% RSLogix 500 project Digital Control.RSS, saved by version 8.30.00.16 %
PROJECT "UNTITLED"    % processor: Bul.1763 MicroLogix 1100 Series B %

PROGRAM FILES
  LAD 2   3 rungs
  LAD 3 "IO"  5 rungs
  LAD 4 "CTRL"  11 rungs

DATA FILES
  O0 OUTPUT  4 elements
  I1 INPUT  6 elements
  S2 STATUS  66 elements
  B3 BINARY  1 elements
  T4 TIMER  4 elements
  C5 COUNTER  1 elements
  R6 CONTROL  1 elements
  N7 INTEGER  1 elements
  F8 FLOAT  1 elements

LADDER 2
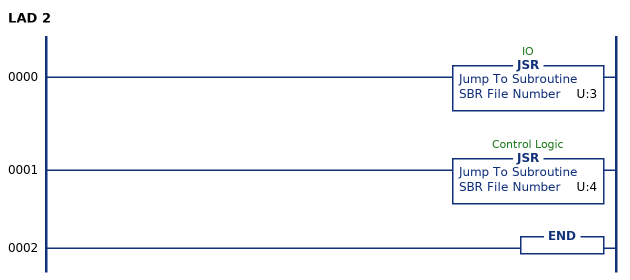
% Rung: 0 %
SOR JSR U:3 EOR
%   U:3  "IO" %
% Rung: 1 %
SOR JSR U:4 EOR
%   U:4  "Control Logic" %
% Rung: 2 %
SOR END EOR

LADDER 3 "IO"
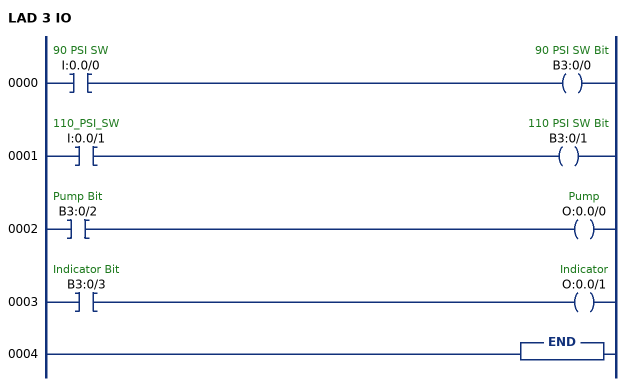
% Rung: 0 %
SOR XIC I:0.0/0 OTE B3:0/0 EOR
%   I:0.0/0  "90 PSI SW" %
%   B3:0/0  "90 PSI SW Bit" %
% Rung: 1 %
SOR XIC I:0.0/1 OTE B3:0/1 EOR
%   I:0.0/1  110_PSI_SW %
%   B3:0/1  "110 PSI SW Bit" %
% Rung: 2 %
SOR XIC B3:0/2 OTE O:0.0/0 EOR
%   B3:0/2  "Pump Bit" %
%   O:0.0/0  "Pump" %
% Rung: 3 %
SOR XIC B3:0/3 OTE O:0.0/1 EOR
%   B3:0/3  "Indicator Bit" %
%   O:0.0/1  "Indicator" %
% Rung: 4 %
SOR END EOR

LADDER 4 "CTRL"
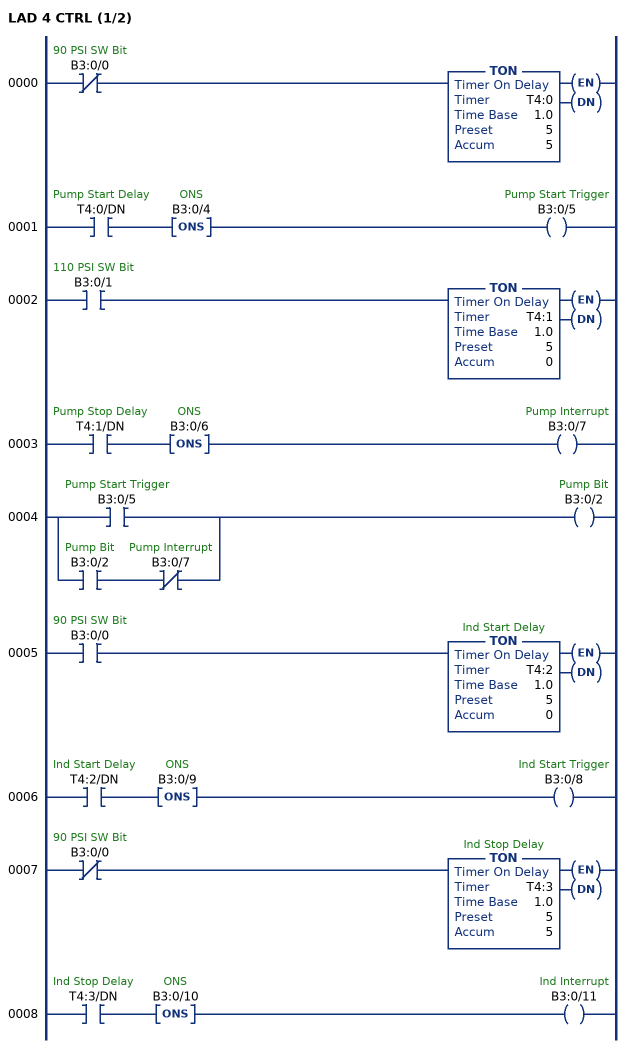
% Rung: 0 %
SOR XIO B3:0/0 TON T4:0 1.0 5 5 EOR
%   B3:0/0  "90 PSI SW Bit" %
% Rung: 1 %
SOR XIC T4:0/DN ONS B3:0/4 OTE B3:0/5 EOR
%   T4:0/DN  "Pump Start Delay" %
%   B3:0/4  "ONS" %
%   B3:0/5  "Pump Start Trigger" %
% Rung: 2 %
SOR XIC B3:0/1 TON T4:1 1.0 5 0 EOR
%   B3:0/1  "110 PSI SW Bit" %
% Rung: 3 %
SOR XIC T4:1/DN ONS B3:0/6 OTE B3:0/7 EOR
%   T4:1/DN  "Pump Stop Delay" %
%   B3:0/6  "ONS" %
%   B3:0/7  "Pump Interrupt" %
% Rung: 4 %
SOR BST XIC B3:0/5 NXB XIC B3:0/2 XIO B3:0/7 BND OTE B3:0/2 EOR
%   B3:0/5  "Pump Start Trigger" %
%   B3:0/2  "Pump Bit" %
%   B3:0/7  "Pump Interrupt" %
% Rung: 5 %
SOR XIC B3:0/0 TON T4:2 1.0 5 0 EOR
%   B3:0/0  "90 PSI SW Bit" %
%   T4:2  "Ind Start Delay" %
% Rung: 6 %
SOR XIC T4:2/DN ONS B3:0/9 OTE B3:0/8 EOR
%   T4:2/DN  "Ind Start Delay" %
%   B3:0/9  "ONS" %
%   B3:0/8  "Ind Start Trigger" %
% Rung: 7 %
SOR XIO B3:0/0 TON T4:3 1.0 5 5 EOR
%   B3:0/0  "90 PSI SW Bit" %
%   T4:3  "Ind Stop Delay" %
% Rung: 8 %
SOR XIC T4:3/DN ONS B3:0/10 OTE B3:0/11 EOR
%   T4:3/DN  "Ind Stop Delay" %
%   B3:0/10  "ONS" %
%   B3:0/11  "Ind Interrupt" %

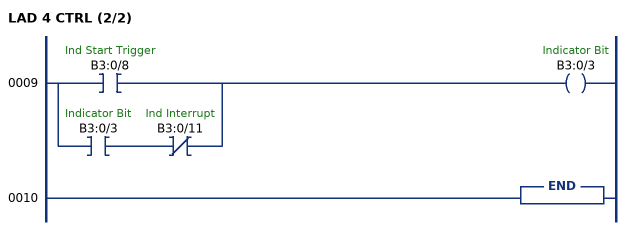
% Rung: 9 %
SOR BST XIC B3:0/8 NXB XIC B3:0/3 XIO B3:0/11 BND OTE B3:0/3 EOR
%   B3:0/8  "Ind Start Trigger" %
%   B3:0/3  "Indicator Bit" %
%   B3:0/11  "Ind Interrupt" %
% Rung: 10 %
SOR END EOR

DATA TABLE (non-zero values as saved)
DATA B3
% B3:0 % 0X0414
DATA T4
% .PRE .ACC %
% T4:0 % 5 5
% T4:1 % 5 0
% T4:2 % 5 0
% T4:3 % 5 5
